INTERFACE I_ActuatorOpenClose EXTENDS I_ActuatorBase

{attribute 'monitoring' := 'call'}
PROPERTY public isClosed : BOOL
GET
END_GET
END_PROPERTY

{attribute 'monitoring' := 'call'}
PROPERTY public isOpened : BOOL
GET
END_GET
END_PROPERTY

METHOD public setClose : BOOL
VAR_INPUT
END_VAR
END_METHOD

METHOD public setOpen : BOOL
VAR_INPUT
END_VAR
END_METHOD

END_INTERFACE

(* stored: Version 1.1.0.1, ProductVersion 3.1.4024.3
   Itf I_ActuatorOpenClose: Id {bd168463-178f-45ac-9d01-7cf59f9ad111}
   Property isClosed: Id {8bcd1611-367e-4f1a-9f22-e0211a266d4b}
   Get Get: Id {8d8e7db6-47ad-4401-b8e9-38f1da3b52cc}
   Property isOpened: Id {97ff894c-3ff8-430a-b82d-5ddf3587aab3}
   Get Get: Id {5f401c41-c682-4bd2-b211-c463625511dd}
   Method setClose: Id {5461888a-4a02-458e-bc56-6c7f1b034c3d}
   Method setOpen: Id {757a091d-ffe9-4f16-9550-33df861752ca} *)
